// TIA Portal V17 export
// export: Created 2025-06-25T13:13:13.7028282Z, ExportSetting WithDefaults, DisplayName Totally Integrated Automation Portal, DisplayVersion V17 Update 8, DisplayName TIA Portal Openness, DisplayVersion V17 Update 8, DisplayName TIA Portal Version Control Interface, DisplayVersion V17, DisplayName STEP 7 Professional, DisplayVersion V17 Update 8, DisplayName STEP 7 Safety, DisplayVersion V17 Update 6, DisplayName WinCC Advanced, DisplayVersion V17 Update 8
FUNCTION_BLOCK "HMI-Communication"   // FB3, FBD
{ S7_Optimized_Access := 'TRUE' }
VERSION : 0.1
// stored: AutoNumber true, IsIECCheckEnabled false, IsRetainMemResEnabled false, MemoryReserve 0, SetENOAutomatically false, UDAEnableTagReadback false
   VAR
      StartRequest : Bool;
      StopRequest : Bool;
      HMI_Running : Bool;
      SkipPauseTime : Bool;
      EmergencyStopWaitTime : Bool;
      SkipEmergencyStopWait : Bool;
      CloseSafetyRelay : Bool;
      OpenSafetyRelay : Bool;
      HMI_Acknowledge_Error : Bool;
      BackToStandby_OilHeat { ExternalVisible := 'False'; ExternalWritable := 'False'} : Bool;
      BackToStandby_SourceFlowNotOK { ExternalVisible := 'False'; ExternalWritable := 'False'} : Bool;
      BackToStandby_SinkFlowNotOK : Bool;
      BackToStandby_SinkTemperatureNotOK : Bool;
      BackToStandby_SourceTemperatureNotOK : Bool;
      BackToStandby_PerformanceControlNotOK : Bool;
      ReturnValvesManualOverride : Bool;   // Hopefully temporary!
      HBL_XV_02override : Bool;   // Temporary!
      HBL_XV_03override : Bool;   // Temporary!
      HBL_HV_860override : Bool;   // Temporary!
      HBL_HV_861override : Bool;   // Temporary!
      State_Text : String;
      BackToStandby_TriggerBit : Bool;   // Bit set if state changes "back to standby"
      BackToStandby_TriggerMemory : Bool;   // Internal flag memory for "back to standby" changes
      BackToStandby_TriggerInt : Int;   // Integer for state changes "back to standby" HMI message
      BackToStandbyReason_Text : String;   // Text to describe "back to standby" reason
      StopReason_TriggerBit : Bool;
      StopReason_TriggerMemory : Bool;
      StopReason_TriggerInt : Int;
      StopReason_Text : String;
      Progress_Text : Int;
      RegulationTarget : Int;
      RegulationTargetPrev : Int;
      HeatboosterSetpoint : Real;   // Main setpoint of the machine
      HeatboosterSetpointPrev : Real;
      EmergencyStopCountdown : Time_Of_Day;
      A1001 { ExternalAccessible := 'False'; ExternalVisible := 'False'; ExternalWritable := 'False'} : "fbHMIEvent";
      WinCCLink { ExternalAccessible := 'False'; ExternalVisible := 'False'; ExternalWritable := 'False'; S7_SetPoint := 'True'} : "fbHeartbeat";
      State2DwellTimeElapsed { S7_SetPoint := 'True'} : Time_Of_Day;
      State2DwellTime : Time_Of_Day;
      State3DwellTimeElapsed : Time_Of_Day;
      State3DwellTime : Time_Of_Day;
      State4DwellTimeElapsed : Time_Of_Day;
      State4DwellTime : Time_Of_Day;
      State5DwellTimeElapsed : Time_Of_Day;
      State5DwellTime : Time_Of_Day;
      State7DwellTimeElapsed : Time_Of_Day;
      State7DwellTime : Time_Of_Day;
      State2PauseTimeElapsed : Time_Of_Day;
      State2PauseTime : Time_Of_Day;
      PurgeControlPurgeTime : Time_Of_Day;
      PurgeControlSpinTime : Time_Of_Day;
      PerformanceControlStandbyTime : Time_Of_Day;
      PerformanceControlStandbyTimeElapsed : Time_Of_Day;
      FilterDryerOnTime : Time_Of_Day;
      FilterDryerOffTime : Time_Of_Day;
      OilRecoveryOnTime : Time_Of_Day;
      ProgressiveTimes : Array[0..3] of Time_Of_Day;
      ProgressiveTime : Time_Of_Day;
      ProgressiveManualTime : Time_Of_Day;
      HV640_OpenTime : Time_Of_Day;
      HV640_CloseTime : Time_Of_Day;
      HV670_OpenTime : Time_Of_Day;
      HV670_CloseTime : Time_Of_Day;
      HV852_OpenTime : Time_Of_Day;
      HV852_CloseTime : Time_Of_Day;
      HV861_OpenTime : Time_Of_Day;
      HV861_CloseTime : Time_Of_Day;
      State2DwellSync { ExternalAccessible := 'False'; ExternalVisible := 'False'; ExternalWritable := 'False'} : "fbWinCCTime";
      State3DwellSync { ExternalAccessible := 'False'; ExternalVisible := 'False'; ExternalWritable := 'False'; S7_SetPoint := 'True'} : "fbWinCCTime";
      State4DwellSync { ExternalAccessible := 'False'; ExternalVisible := 'False'; ExternalWritable := 'False'; S7_SetPoint := 'True'} : "fbWinCCTime";
      State5DwellSync { ExternalAccessible := 'False'; ExternalVisible := 'False'; ExternalWritable := 'False'; S7_SetPoint := 'True'} : "fbWinCCTime";
      State7DwellSync { ExternalAccessible := 'False'; ExternalVisible := 'False'; ExternalWritable := 'False'; S7_SetPoint := 'True'} : "fbWinCCTime";
      State2PauseSync { ExternalAccessible := 'False'; ExternalVisible := 'False'; ExternalWritable := 'False'; S7_SetPoint := 'True'} : "fbWinCCTime";
      PurgeControlPurgeSync { ExternalAccessible := 'False'; ExternalVisible := 'False'; ExternalWritable := 'False'; S7_SetPoint := 'True'} : "fbWinCCTime";
      PurgeControlSpinSync { ExternalAccessible := 'False'; ExternalVisible := 'False'; ExternalWritable := 'False'; S7_SetPoint := 'True'} : "fbWinCCTime";
      ProgressiveTime0Sync { ExternalAccessible := 'False'; ExternalVisible := 'False'; ExternalWritable := 'False'; S7_SetPoint := 'True'} : "fbWinCCTime";
      ProgressiveTime1Sync { ExternalAccessible := 'False'; ExternalVisible := 'False'; ExternalWritable := 'False'; S7_SetPoint := 'True'} : "fbWinCCTime";
      ProgressiveTime2Sync { ExternalAccessible := 'False'; ExternalVisible := 'False'; ExternalWritable := 'False'; S7_SetPoint := 'True'} : "fbWinCCTime";
      ProgressiveTime3Sync { ExternalAccessible := 'False'; ExternalVisible := 'False'; ExternalWritable := 'False'; S7_SetPoint := 'True'} : "fbWinCCTime";
      ProgressiveManualTimeSync { ExternalAccessible := 'False'; ExternalVisible := 'False'; ExternalWritable := 'False'; S7_SetPoint := 'True'} : "fbWinCCTime";
      PerformanceControlStandbySync { ExternalAccessible := 'False'; ExternalVisible := 'False'; ExternalWritable := 'False'; S7_SetPoint := 'True'} : "fbWinCCTime";
      FilterDryerOnTimeSync { S7_SetPoint := 'True'} : "fbWinCCTime";
      FilterDryerOffTimeSync { S7_SetPoint := 'True'} : "fbWinCCTime";
      OilRecoveryOnTimeSync { S7_SetPoint := 'True'} : "fbWinCCTime";
      HV640_OpenTimeSync { S7_SetPoint := 'True'} : "fbWinCCTime";
      HV640_CloseTimeSync { S7_SetPoint := 'True'} : "fbWinCCTime";
      HV670_OpenTimeSync { S7_SetPoint := 'True'} : "fbWinCCTime";
      HV670_CloseTimeSync { S7_SetPoint := 'True'} : "fbWinCCTime";
      HV852_OpenTimeSync { S7_SetPoint := 'True'} : "fbWinCCTime";
      HV852_CloseTimeSync { S7_SetPoint := 'True'} : "fbWinCCTime";
      HV861_OpenTimeSync { S7_SetPoint := 'True'} : "fbWinCCTime";
      HV861_CloseTimeSync { S7_SetPoint := 'True'} : "fbWinCCTime";
   END_VAR
   VAR_TEMP
      FellBackToStandby_456 : Bool;
      FellBackToStandby_56 : Bool;
   END_VAR
   VAR CONSTANT
      "01_WaitingForStateChange" : SInt := 1;
      "02_ErrorAcknowledge" : SInt := 2;
      "03_SafetyRelayNotClosed" : SInt := 3;
      "04_SafetyRelayInterrupted" : SInt := 4;
      "05_CPU_Init" : SInt := 5;
      "6_CriticalAlarmActive" : SInt := 6;
      "10_ReadyToStart" : SInt := 10;
      "11_EmergencyStopActive" : SInt := 11;
      "12_InverterNotOnline" : SInt := 12;
      "13_ReadyToStartWithActiveWarnings" : SInt := 13;
      "14_EmergencyStopWaitTime" : SInt := 14;
      "20_WaitForSourceFlow" : SInt := 20;
      "21_WaitForSinkFlow" : SInt := 21;
      "22_WaitForSinkHeat" : SInt := 22;
      "23_WaitForSourceHeat" : SInt := 23;
      "24_PauseTime" : SInt := 24;
      "25_PowerControlZeroperformanceDemand" : SInt := 25;
      "26_HeatSink_Limit" : SInt := 26;
      "27_HeatSource_Limit" : SInt := 27;
      "28_VariableControl_Limit" : SInt := 28;
      "29_WaitingForShaftSeal" : SInt := 29;
      "210_State2DwellTime" : Int := 210;
      "30_PerformanceControlNotReady" : SInt := 30;
      "31_LubricationPrimingNotReady" : SInt := 31;
      "39_State3DwellTime" : SInt := 39;
      "50_WaitForOilHeat" : SInt := 50;
      "51_RampingUp" : SInt := 51;
      "52_DryingSuctionLine" : SInt := 52;
      "53_WaitForSuperHeatOut" : SInt := 53;
      "54_WaitForRecuperator" : SInt := 54;
      "55_SuctionManifoldPurge" : SInt := 55;
      "56_StartingAndHydrolock" : SInt := 56;
      "59_State4DwellTime" : SInt := 59;
      "60_Running" : SInt := 60;
      "61_State5DwellTime" : SInt := 61;
      "62_RunningAndHydrolock" : SInt := 62;
      "70_Stopping" : SInt := 70;
      "71_State7DwellTime" : SInt := 71;
      "72_StoppingDrySuctionLine" : SInt := 72;
      "302_PausedInState2" : Int := 302;
      "303_PausedInState3" : Int := 303;
      "304_PausedInState4" : Int := 304;
      "305_PausedInState5" : Int := 305;
      "307_PausedInState7" : Int := 307;
   END_VAR
   VAR_TEMP   // added for the SCL form of the ladder/FBD networks
      _w1 : Bool;
      _w2 : Bool;
   END_VAR
BEGIN

REGION Network 1 (SCL): Comments
   (* 
   What's with the fbWinCCTime & Time_Of_Day variables?

   When WinCC displays a TIME variable, it shows it as an integer number of milliseconds. So 5 minutes is 300,000ms. Not very intutive. 
   For longer times, like 1h20min, it's 4,800,000ms. To get a nice display of HH:MM:SS on the screen, and be able to enter time in this 
   format also, the Time_Of_Day variable type has to be used.

   All regulators & other structs use TIME because it's the right type to use, and the same is used everywhere for uniformity. WinCC 
   requires Time_Of_Day for usability. So instead of wrecking the structure and regularity of all those beautiful structs, a conversion 
   is done here (from TIME to TOD and back) to make TIME values "just work" in WinCC. It's ugly but it works, and frees the structs to be
   made the way the design requires, not the way WinCC requires.
   *)
END_REGION

REGION Network 2: Heartbeat
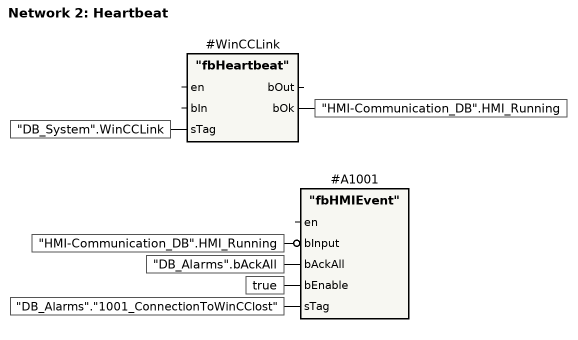
   #WinCCLink(sTag := "DB_System".WinCCLink, bOk => "HMI-Communication_DB".HMI_Running);   // "fbHeartbeat"
   #A1001(bInput := NOT "HMI-Communication_DB".HMI_Running,   // "fbHMIEvent"
          bAckAll := "DB_Alarms".bAckAll,
          bEnable := true,
          sTag := "DB_Alarms"."1001_ConnectionToWinCClost");
END_REGION

REGION Network 3: BackToStandby reason logic
   // Function to show, why the process fell back to standby
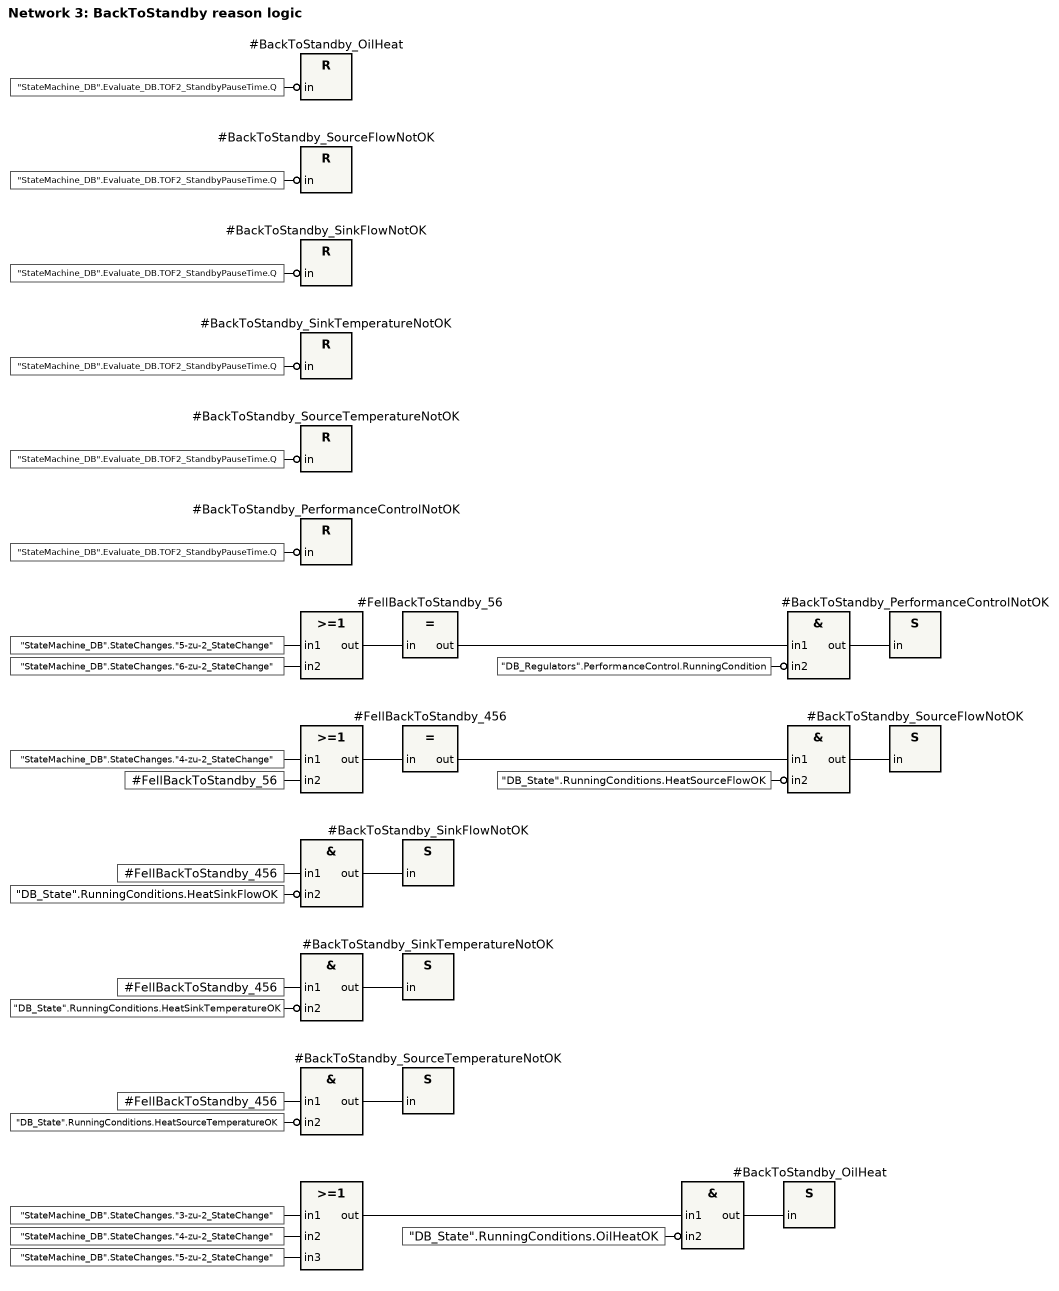
   IF NOT "StateMachine_DB".Evaluate_DB.TOF2_StandbyPauseTime.Q THEN
       #BackToStandby_OilHeat := FALSE;
       #BackToStandby_SourceFlowNotOK := FALSE;
       #BackToStandby_SinkFlowNotOK := FALSE;
       #BackToStandby_SinkTemperatureNotOK := FALSE;
       #BackToStandby_SourceTemperatureNotOK := FALSE;
       #BackToStandby_PerformanceControlNotOK := FALSE;
   END_IF;
   #FellBackToStandby_56 := "StateMachine_DB".StateChanges."5-zu-2_StateChange" OR "StateMachine_DB".StateChanges."6-zu-2_StateChange";
   IF #FellBackToStandby_56 AND NOT "DB_Regulators".PerformanceControl.RunningCondition THEN
       #BackToStandby_PerformanceControlNotOK := TRUE;
   END_IF;
   #FellBackToStandby_456 := "StateMachine_DB".StateChanges."4-zu-2_StateChange" OR #FellBackToStandby_56;
   IF #FellBackToStandby_456 AND NOT "DB_State".RunningConditions.HeatSourceFlowOK THEN
       #BackToStandby_SourceFlowNotOK := TRUE;
   END_IF;
   IF #FellBackToStandby_456 AND NOT "DB_State".RunningConditions.HeatSinkFlowOK THEN
       #BackToStandby_SinkFlowNotOK := TRUE;
   END_IF;
   IF #FellBackToStandby_456 AND NOT "DB_State".RunningConditions.HeatSinkTemperatureOK THEN
       #BackToStandby_SinkTemperatureNotOK := TRUE;
   END_IF;
   IF #FellBackToStandby_456 AND NOT "DB_State".RunningConditions.HeatSourceTemperatureOK THEN
       #BackToStandby_SourceTemperatureNotOK := TRUE;
   END_IF;
   IF ("StateMachine_DB".StateChanges."3-zu-2_StateChange" OR "StateMachine_DB".StateChanges."4-zu-2_StateChange" OR "StateMachine_DB".StateChanges."5-zu-2_StateChange") AND NOT "DB_State".RunningConditions.OilHeatOK THEN
       #BackToStandby_OilHeat := TRUE;
   END_IF;
END_REGION

REGION Network 4: BackToStandby-bit to trigger HMI-Message
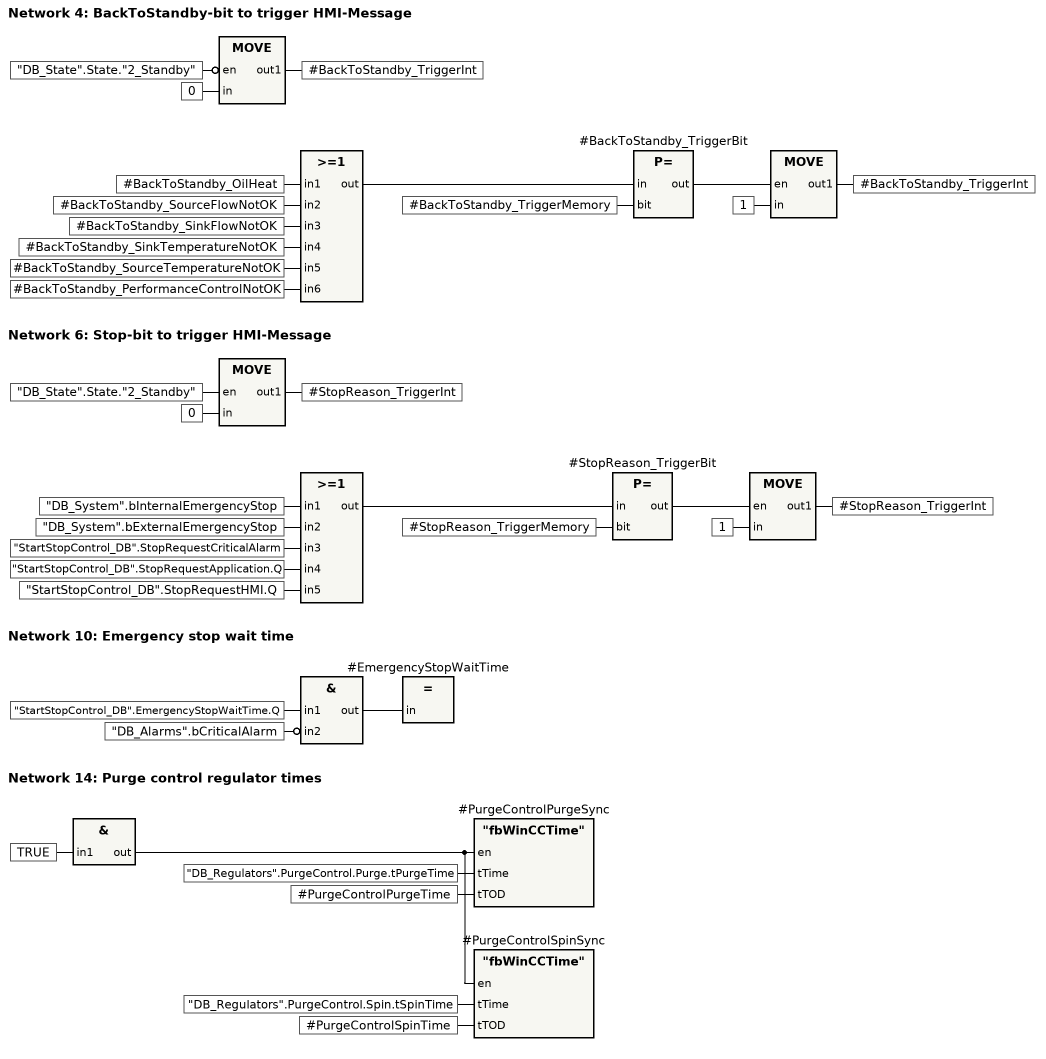
   IF NOT "DB_State".State."2_Standby" THEN #BackToStandby_TriggerInt := 0; END_IF;
   #_w1 := #BackToStandby_OilHeat OR #BackToStandby_SourceFlowNotOK OR #BackToStandby_SinkFlowNotOK OR #BackToStandby_SinkTemperatureNotOK OR #BackToStandby_SourceTemperatureNotOK OR #BackToStandby_PerformanceControlNotOK;
   #BackToStandby_TriggerBit := #_w1 AND NOT #BackToStandby_TriggerMemory;   // rising edge
   #BackToStandby_TriggerMemory := #_w1;
   IF #_w1 THEN #BackToStandby_TriggerInt := 1; END_IF;
END_REGION

REGION Network 5 (SCL): BackToStandby reason text
   // Write "back-to-standby" reason to text and deliver it to the HMI
   IF #BackToStandby_OilHeat THEN
       #BackToStandbyReason_Text := 'Oil heat was not OK!';
   ELSIF #BackToStandby_PerformanceControlNotOK THEN
       #BackToStandbyReason_Text := 'No power was required!';
   ELSIF #BackToStandby_SourceTemperatureNotOK THEN
       #BackToStandbyReason_Text := 'Heat source was not OK!';
   ELSIF #BackToStandby_SinkTemperatureNotOK THEN
       #BackToStandbyReason_Text := 'Heat sink was not OK!';
   ELSIF #BackToStandby_SourceFlowNotOK THEN
       #BackToStandbyReason_Text := 'No source mass flow!';
   ELSIF #BackToStandby_SinkFlowNotOK THEN
       #BackToStandbyReason_Text := 'No sink mass flow!';
   ELSE
       #BackToStandbyReason_Text := '';
   END_IF;
END_REGION

REGION Network 6: Stop-bit to trigger HMI-Message
   IF "DB_State".State."2_Standby" THEN #StopReason_TriggerInt := 0; END_IF;
   #_w1 := "DB_System".bInternalEmergencyStop OR "DB_System".bExternalEmergencyStop OR "StartStopControl_DB".StopRequestCriticalAlarm OR "StartStopControl_DB".StopRequestApplication.Q OR "StartStopControl_DB".StopRequestHMI.Q;
   #StopReason_TriggerBit := #_w1 AND NOT #StopReason_TriggerMemory;   // rising edge
   #StopReason_TriggerMemory := #_w1;
   IF #_w1 THEN #StopReason_TriggerInt := 1; END_IF;
END_REGION

REGION Network 7 (SCL): Stop reason text
   // Write stop reason to text and deliver it to the HMI
   IF "DB_System".bInternalEmergencyStop THEN
       //Emergency Stop intern
       #StopReason_Text := 'Internal emergency stopp!';
   ELSIF "DB_System".bExternalEmergencyStop THEN
       //Emergency Stop extern
       #StopReason_Text := 'External emergency stopp!';
   ELSIF "StartStopControl_DB".StopRequestCriticalAlarm THEN
       //Stop via critical alarm 
       #StopReason_Text := 'Critical alarm!';
   ELSIF "StartStopControl_DB".StopRequestApplication.Q THEN
       //Stop via application PLC
       #StopReason_Text := 'External stopp request!';
   ELSIF "StartStopControl_DB".StopRequestHMI.Q THEN
       //Stop via HMI  
       #StopReason_Text := 'HMI stopp request!';
   END_IF;
END_REGION

REGION Network 8 (SCL): State text & progress text
   // #Progress_Text = 1 is the catch-all error state. If you end up there then there is more work to do.
   CASE "DB_State".State.State_Number OF
       0:  #State_Text := 'Init';

           IF "DB_State".SystemInitialised = FALSE THEN
               #Progress_Text := #"05_CPU_Init";
           ELSE
               #Progress_Text := #"01_WaitingForStateChange";
           END_IF;

       1:  #State_Text := 'Offline';

           IF "DB_System".bEmergencyStop = TRUE THEN
               #Progress_Text := #"11_EmergencyStopActive";
           ELSIF "DB_Alarms"."1110_HBL_SC_10_CommError".sState.bActive OR "DB_Alarms"."1130_HBL_SC_10_Tripped".sState.bActive THEN
               #Progress_Text := #"12_InverterNotOnline";
           ELSIF "DB_Alarms".bCriticalAlarm = TRUE THEN
               #Progress_Text := #"6_CriticalAlarmActive";
           ELSIF "StartStopControl_DB".EmergencyStopWaitTime.Q = TRUE THEN
               #Progress_Text := #"14_EmergencyStopWaitTime";
           ELSIF "DB_Alarms".bCommonAlarm = TRUE THEN
               #Progress_Text := #"13_ReadyToStartWithActiveWarnings";
           ELSE
               #Progress_Text := #"10_ReadyToStart";
           END_IF;


       2:  #State_Text := 'Standby';

           IF "DB_State".RunningConditions.HeatSourceFlowOK = FALSE THEN
               #Progress_Text := #"20_WaitForSourceFlow";
           ELSIF "DB_State".RunningConditions.HeatSinkFlowOK = FALSE THEN
               #Progress_Text := #"21_WaitForSinkFlow";
           ELSIF "DB_State".RunningConditions.HeatSinkTemperatureOK = FALSE THEN
               #Progress_Text := #"22_WaitForSinkHeat";
           ELSIF "DB_State".RunningConditions.HeatSourceTemperatureOK = FALSE THEN
               #Progress_Text := #"23_WaitForSourceHeat";
           ELSIF "StateMachine_DB".Evaluate_DB.TOF2_StandbyPauseTime.Q = TRUE THEN
               #Progress_Text := #"24_PauseTime";
           ELSIF "StateMachine_DB".Evaluate_DB.TON2_Standby.Q = FALSE THEN
               #Progress_Text :=#"210_State2DwellTime";
           ELSIF "DB_Regulators".PerformanceControl.RunningCondition = FALSE THEN
               IF "Regulation_DB".PerformanceControl.HeatSinkTimer.Q = FALSE THEN
                   #Progress_Text := #"26_HeatSink_Limit";
               ELSIF ("Regulation_DB".PerformanceControl.HeatSourceTimer.Q) = FALSE THEN
                   #Progress_Text := #"27_HeatSource_Limit";
               ELSIF "Regulation_DB".PerformanceControl.VariableControlTimer.Q = FALSE THEN
                   #Progress_Text := #"28_VariableControl_Limit";
               ELSE
                   #Progress_Text := #"25_PowerControlZeroperformanceDemand";
               END_IF;
           ELSIF "DB_State".StatePauseFlags[2] = TRUE THEN
               #Progress_Text := #"302_PausedInState2";
           ELSE
               #Progress_Text := #"01_WaitingForStateChange";
           END_IF;

       3:  #State_Text := 'Prepare Start';

           IF "DB_State".RunningConditions.ShaftSealSystemOK = FALSE THEN
               #Progress_Text := #"29_WaitingForShaftSeal";
           ELSIF "DB_State".RunningConditions.OilHeatOK = FALSE THEN
               #Progress_Text := #"50_WaitForOilHeat";
           ELSIF "DB_State".RunningConditions.LubricationPrimingOk = FALSE THEN
               #Progress_Text := #"31_LubricationPrimingNotReady";
           ELSIF "DB_Regulators".PerformanceControl.RunningCondition = FALSE THEN
               #Progress_Text := #"30_PerformanceControlNotReady";
           ELSIF "StateMachine_DB".Evaluate_DB.TON3_PrepareStart.Q = FALSE THEN
               #Progress_Text := #"39_State3DwellTime";
           ELSIF "DB_State".StatePauseFlags[3] = TRUE THEN
               #Progress_Text := #"303_PausedInState3";
           ELSE
               #Progress_Text := #"01_WaitingForStateChange";
           END_IF;

       4:  #State_Text := 'Starting';

           IF "DB_State".RunningConditions.DoWarmStart = FALSE AND "DB_Regulators".PurgeControl.bDone = FALSE THEN
               #Progress_Text := #"55_SuctionManifoldPurge";
           ELSIF "DB_State".RunningConditions.AtOrAboveHydrolockSpeed = FALSE THEN
               #Progress_Text := #"51_RampingUp";
           ELSIF "DB_State".RunningConditions.SuctionLineDry = FALSE THEN
               #Progress_Text := #"52_DryingSuctionLine";
           ELSIF "StateMachine_DB".Evaluate_DB.TON4_Start.Q = FALSE THEN
               #Progress_Text := #"59_State4DwellTime";
           ELSIF "DB_State".StatePauseFlags[4] = TRUE THEN
               #Progress_Text := #"304_PausedInState4";
           ELSE
               #Progress_Text := #"01_WaitingForStateChange";
           END_IF;

       5:  #State_Text := 'Warm-up';

           IF "DB_State".RunningConditions.RiskOfHydrolock = TRUE THEN
               #Progress_Text := #"56_StartingAndHydrolock";
           ELSIF "DB_State".RunningConditions.SuperheatCompressorOutOK = FALSE THEN
               #Progress_Text := #"53_WaitForSuperHeatOut";
           ELSIF "DB_State".RunningConditions.RecuperatorWorking = FALSE THEN
               #Progress_Text := #"54_WaitForRecuperator";
           ELSIF "StateMachine_DB".Evaluate_DB.TON5_Warmup.Q = FALSE THEN
               #Progress_Text := #"61_State5DwellTime";
           ELSIF "DB_State".StatePauseFlags[5] = TRUE THEN
               #Progress_Text := #"305_PausedInState5";
           ELSE
               #Progress_Text := #"01_WaitingForStateChange";
           END_IF;

       6:  #State_Text := 'Running';
           IF "DB_State".RunningConditions.RiskOfHydrolock = TRUE THEN
               #Progress_Text := #"62_RunningAndHydrolock";
           ELSE
               #Progress_Text := #"60_Running";
           END_IF;

       7:  #State_Text := 'Stop';

           IF "DB_State".RunningConditions.SuctionLineDry = FALSE AND"DB_State".FastStop = FALSE THEN
               #Progress_Text := #"72_StoppingDrySuctionLine";
           ELSIF "DB_InverterDrives".HBL_SC_10.Stat.Speed.Eng.fValue <> 0 THEN
               #Progress_Text := #"70_Stopping";
           ELSIF "StateMachine_DB".Evaluate_DB.TON7_Stop.Q = FALSE THEN
               #Progress_Text := #"71_State7DwellTime";
           ELSE
               #Progress_Text := #"01_WaitingForStateChange";
           END_IF;

       ELSE  
           #State_Text := 'No state!';
   END_CASE;
END_REGION

REGION Network 9 (SCL): Regulation target
   // Repeating some of the logic from PerformanceControl (FB9) here, making it fragile
   // Conditions are evaluated as repeated IFs and not ELSIFs because that is how it is evaluated in FB9. Yes, confusing.
   // This network provides an alternative interface to Performance Control, using its public API (DB_Regulators.PerformanceControl)
   // Figure out which target is active & select setpoint
   IF "DB_Regulators".PerformanceControl.Settings.HeatSink.Control_Active THEN
       IF "DB_Regulators".PerformanceControl.Settings.HeatSink.UseFeedFlow THEN
           #RegulationTarget := 2;
       ELSE
           #RegulationTarget := 1;
       END_IF;
   END_IF;

   IF "DB_Regulators".PerformanceControl.Settings.HeatSource.Control_Active THEN
       IF "DB_Regulators".PerformanceControl.Settings.HeatSource.UseFeedFlow THEN
           #RegulationTarget := 4;
       ELSE
           #RegulationTarget := 3;
       END_IF;
   END_IF;

   IF "DB_Regulators".PerformanceControl.Settings.VariableControl.Control_Active AND "DB_Regulators".PerformanceControl.Settings.VariableControl.ReferenceID > 0 THEN
       #RegulationTarget := 6;
   END_IF;

   // Update the currently selected setpoint if updated from HMI
   IF #HeatboosterSetpoint <> #HeatboosterSetpointPrev THEN
       // Select the right setpoint
       CASE #RegulationTarget OF
       1..2 : "DB_Regulators".PerformanceControl.Settings.HeatSink.Setpoint := #HeatboosterSetpoint;
       3..4 : "DB_Regulators".PerformanceControl.Settings.HeatSource.Setpoint := #HeatboosterSetpoint;
       6    : "DB_Regulators".PerformanceControl.Settings.VariableControl.Setpoint := #HeatboosterSetpoint;
       END_CASE;
   END_IF;
   #HeatboosterSetpointPrev := #HeatboosterSetpoint;
END_REGION

REGION Network 10: Emergency stop wait time
   // Do not show when a critical alarm is active
   #EmergencyStopWaitTime := "StartStopControl_DB".EmergencyStopWaitTime.Q AND NOT "DB_Alarms".bCriticalAlarm;
END_REGION

REGION Network 11 (SCL): Emergency lock time
   // Gruesome, this needs refactoring
   #EmergencyStopCountdown := TIME_TO_TOD(IN := ("StartStopControl_DB".EmergencyStopWaitTime.PT - "StartStopControl_DB".EmergencyStopWaitTime.ET));
   IF #SkipEmergencyStopWait THEN
       RESET_TIMER("StartStopControl_DB".EmergencyStopWaitTime);
   END_IF;
END_REGION

REGION Network 12 (SCL): Dwell times
   #State2DwellTimeElapsed := TIME_TO_TOD("StateMachine_DB".Evaluate_DB.TON2_Standby.ET);
   #State2DwellSync(tTime := "DB_CurrentSetting".MissingSetting.Misc.State2DwellTime, tTOD := #State2DwellTime);

   #State3DwellTimeElapsed := TIME_TO_TOD("StateMachine_DB".Evaluate_DB.TON3_PrepareStart.ET);
   #State3DwellSync(tTime := "DB_CurrentSetting".MissingSetting.Misc.State3DwellTime, tTOD := #State3DwellTime);

   #State4DwellTimeElapsed := TIME_TO_TOD("StateMachine_DB".Evaluate_DB.TON4_Start.ET);
   #State4DwellSync(tTime := "DB_CurrentSetting".MissingSetting.Misc.State4DwellTime, tTOD := #State4DwellTime);

   #State5DwellTimeElapsed := TIME_TO_TOD("StateMachine_DB".Evaluate_DB.TON5_Warmup.ET);
   #State5DwellSync(tTime := "DB_CurrentSetting".MissingSetting.Misc.State5DwellTime, tTOD := #State5DwellTime);

   #State7DwellTimeElapsed := TIME_TO_TOD("StateMachine_DB".Evaluate_DB.TON7_Stop.ET);
   #State7DwellSync(tTime := "DB_CurrentSetting".MissingSetting.Misc.State7DwellTime, tTOD := #State7DwellTime);
END_REGION

REGION Network 13 (SCL): Pause time
   #State2PauseTimeElapsed := TIME_TO_TOD("StateMachine_DB".Evaluate_DB.TOF2_StandbyPauseTime.ET);
   #State2PauseSync(tTime := "DB_CurrentSetting".MissingSetting.Misc.State2PauseTime, tTOD := #State2PauseTime);
END_REGION

REGION Network 14: Purge control regulator times
   IF TRUE THEN
       #PurgeControlPurgeSync(tTime := "DB_Regulators".PurgeControl.Purge.tPurgeTime,   // "fbWinCCTime"
                              tTOD := #PurgeControlPurgeTime);
       #PurgeControlSpinSync(tTime := "DB_Regulators".PurgeControl.Spin.tSpinTime, tTOD := #PurgeControlSpinTime);   // "fbWinCCTime"
   END_IF;
END_REGION

REGION Network 15: CPC progressive regulator
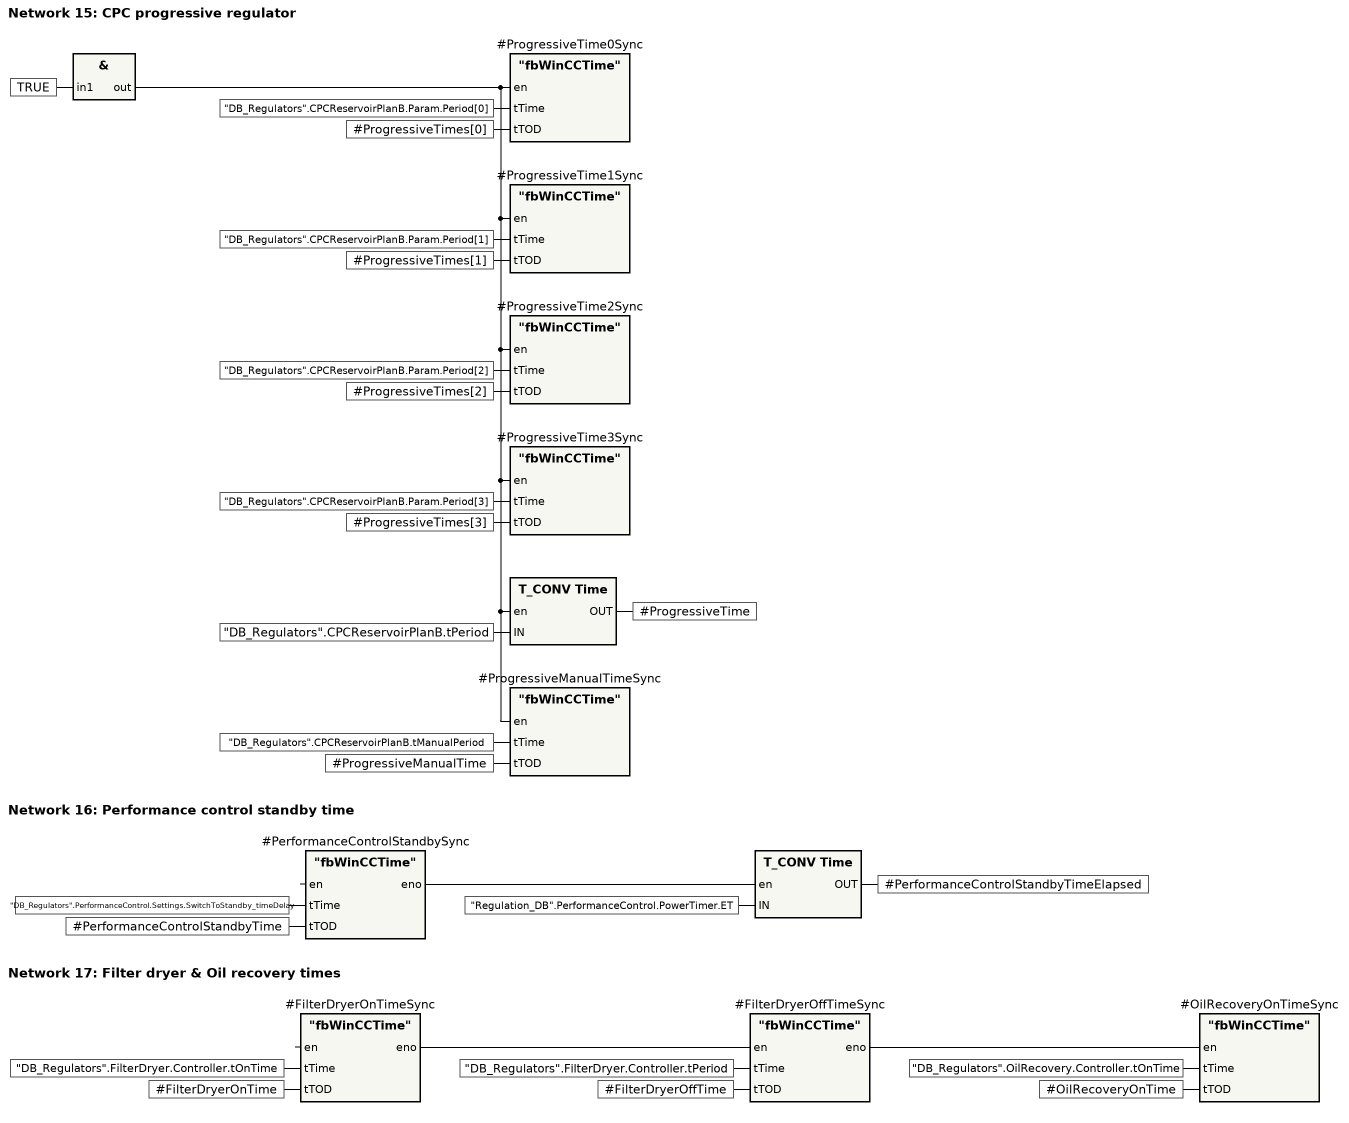
   IF TRUE THEN
       #ProgressiveTime0Sync(tTime := "DB_Regulators".CPCReservoirPlanB.Param.Period[0],   // "fbWinCCTime"
                             tTOD := #ProgressiveTimes[0]);
       #ProgressiveTime1Sync(tTime := "DB_Regulators".CPCReservoirPlanB.Param.Period[1],   // "fbWinCCTime"
                             tTOD := #ProgressiveTimes[1]);
       #ProgressiveTime2Sync(tTime := "DB_Regulators".CPCReservoirPlanB.Param.Period[2],   // "fbWinCCTime"
                             tTOD := #ProgressiveTimes[2]);
       #ProgressiveTime3Sync(tTime := "DB_Regulators".CPCReservoirPlanB.Param.Period[3],   // "fbWinCCTime"
                             tTOD := #ProgressiveTimes[3]);
       T_CONV(IN := "DB_Regulators".CPCReservoirPlanB.tPeriod, OUT => #ProgressiveTime);
       #ProgressiveManualTimeSync(tTime := "DB_Regulators".CPCReservoirPlanB.tManualPeriod,   // "fbWinCCTime"
                               tTOD := #ProgressiveManualTime);
   END_IF;
END_REGION

REGION Network 16: Performance control standby time
   #PerformanceControlStandbySync(tTime := "DB_Regulators".PerformanceControl.Settings.SwitchToStandby_timeDelay,   // "fbWinCCTime"
                           tTOD := #PerformanceControlStandbyTime,
                           ENO => #_w1);
   IF #_w1 THEN
       T_CONV(IN := "Regulation_DB".PerformanceControl.PowerTimer.ET, OUT => #PerformanceControlStandbyTimeElapsed);
   END_IF;
END_REGION

REGION Network 17: Filter dryer & Oil recovery times
   #FilterDryerOnTimeSync(tTime := "DB_Regulators".FilterDryer.Controller.tOnTime,   // "fbWinCCTime"
                          tTOD := #FilterDryerOnTime,
                          ENO => #_w1);
   #FilterDryerOffTimeSync(EN := #_w1,   // "fbWinCCTime"
                           tTime := "DB_Regulators".FilterDryer.Controller.tPeriod,
                           tTOD := #FilterDryerOffTime,
                           ENO => #_w2);
   IF #_w2 THEN
       #OilRecoveryOnTimeSync(tTime := "DB_Regulators".OilRecovery.Controller.tOnTime, tTOD := #OilRecoveryOnTime);   // "fbWinCCTime"
   END_IF;
END_REGION

REGION Network 18: Process Valves
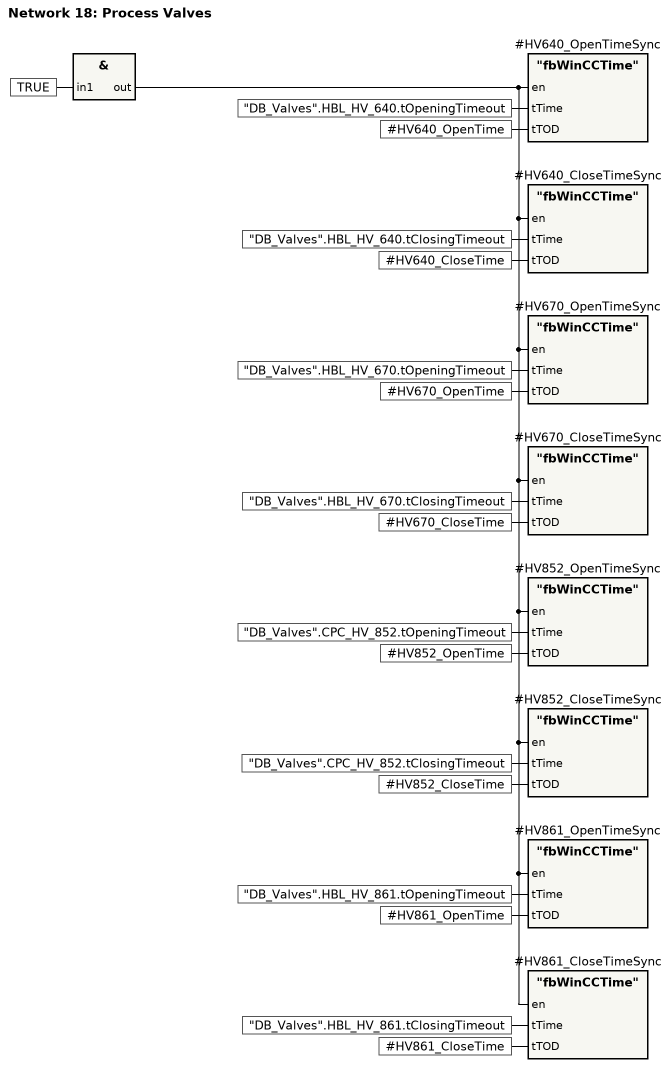
   IF TRUE THEN
       #HV640_OpenTimeSync(tTime := "DB_Valves".HBL_HV_640.tOpeningTimeout, tTOD := #HV640_OpenTime);   // "fbWinCCTime"
       #HV640_CloseTimeSync(tTime := "DB_Valves".HBL_HV_640.tClosingTimeout, tTOD := #HV640_CloseTime);   // "fbWinCCTime"
       #HV670_OpenTimeSync(tTime := "DB_Valves".HBL_HV_670.tOpeningTimeout, tTOD := #HV670_OpenTime);   // "fbWinCCTime"
       #HV670_CloseTimeSync(tTime := "DB_Valves".HBL_HV_670.tClosingTimeout, tTOD := #HV670_CloseTime);   // "fbWinCCTime"
       #HV852_OpenTimeSync(tTime := "DB_Valves".CPC_HV_852.tOpeningTimeout, tTOD := #HV852_OpenTime);   // "fbWinCCTime"
       #HV852_CloseTimeSync(tTime := "DB_Valves".CPC_HV_852.tClosingTimeout, tTOD := #HV852_CloseTime);   // "fbWinCCTime"
       #HV861_OpenTimeSync(tTime := "DB_Valves".HBL_HV_861.tOpeningTimeout, tTOD := #HV861_OpenTime);   // "fbWinCCTime"
       #HV861_CloseTimeSync(tTime := "DB_Valves".HBL_HV_861.tClosingTimeout, tTOD := #HV861_CloseTime);   // "fbWinCCTime"
   END_IF;
END_REGION
END_FUNCTION_BLOCK
